// TIA Portal V15.1 export
// export: Created 2024-06-21T08:40:42.5093779Z, ExportSetting WithDefaults, DisplayName Totally Integrated Automation Portal, DisplayVersion V15.1 Update 5, DisplayName TIA Portal Openness, DisplayVersion V15.1 Update 5, DisplayName SINAMICS Startdrive Advanced, DisplayVersion V15.1, DisplayName G130, G150, S120, S150, SINAMICS MV, S210, DisplayVersion V15.1, DisplayName G110M, G120, G120C, G120D, G120P, DisplayVersion V15.1, DisplayName STEP 7 Professional, DisplayVersion V15.1 Update 5, DisplayName STEP 7 Safety, DisplayVersion V15.1, DisplayName WinCC Professional, DisplayVersion V15.1 Update 5, DisplayName SIMATIC Visualization Architect, DisplayVersion V15.1
DATA_BLOCK "_209000NCP01PNIODiag"   // DB270
{ S7_Optimized_Access := 'FALSE' }
AUTHOR : VCC
VERSION : 0.1
// stored: AutoNumber false, DBAccessibleFromOPCUA true, IsOnlyStoredInLoadMemory false, IsWriteProtectedInAS false
   VAR RETAIN
      "AD_209000AK01E1-BE30" { ExternalAccessible := 'False'; ExternalVisible := 'False'; ExternalWritable := 'False'} : Bool;   // Profinet device doesn't exist - PAC - Cabinet AK01 - node 30
      "AC_209000AE01-JC31" { ExternalAccessible := 'False'; ExternalVisible := 'False'; ExternalWritable := 'False'} : Bool;   // Profinet device doesn't exist - Gateway ETA Fuse - Cabinet AE01 - node 31
      "AC_209000AK02-JC32" { ExternalAccessible := 'False'; ExternalVisible := 'False'; ExternalWritable := 'False'} : Bool;   // Profinet device doesn't exist - Gateway ETA Fuse - Cabinet AK02 - node 32
      "AA_209000AK01-JW35" { ExternalAccessible := 'False'; ExternalVisible := 'False'; ExternalWritable := 'False'} : Bool;   // Profinet device doesn't exist - ET200sp I/O - Busnode AK01 - node 35
      "AA_209000AK03-JW36" { ExternalAccessible := 'False'; ExternalVisible := 'False'; ExternalWritable := 'False'} : Bool;   // Profinet device doesn't exist - ET200sp I/O - Busnode AK03 - node 36
      "AA_209000AK04-JW37" { ExternalAccessible := 'False'; ExternalVisible := 'False'; ExternalWritable := 'False'} : Bool;   // Profinet device doesn't exist - ET200sp I/O - Busnode AK04 - node 37
      "AA_209000AS01-JW38" { ExternalAccessible := 'False'; ExternalVisible := 'False'; ExternalWritable := 'False'} : Bool;   // Profinet device doesn't exist - ET200sp I/O - Busnode AS01 - node 38
      "AA_209000AS02-JW39" { ExternalAccessible := 'False'; ExternalVisible := 'False'; ExternalWritable := 'False'} : Bool;   // Profinet device doesn't exist - ET200sp I/O - Busnode AS02 - node 39
      "AA_209000AE02-JW208" { ExternalAccessible := 'False'; ExternalVisible := 'False'; ExternalWritable := 'False'} : Bool;   // Profinet device doesn't exist - PN/PN coupler - 209000 <-> 308210 AE02 - node 208
      "AA_209000AE02-JW210" { ExternalAccessible := 'False'; ExternalVisible := 'False'; ExternalWritable := 'False'} : Bool;   // Profinet device doesn't exist - Switch - Cabinet AE02 - node 210
      "AA_209000AE02-JW211" { ExternalAccessible := 'False'; ExternalVisible := 'False'; ExternalWritable := 'False'} : Bool;   // Profinet device doesn't exist - Switch - Cabinet AE02 - node 211
      "AA_211212AE1-JW200" { ExternalAccessible := 'False'; ExternalVisible := 'False'; ExternalWritable := 'False'} : Bool;   // Profinet device doesn't exist - ET200sp I/O - Busnode PLS211212AE1 - node 200
      "AC_209000AK01E1-BE30Fault" { ExternalAccessible := 'False'; ExternalVisible := 'False'; ExternalWritable := 'False'} : Bool;   // Faulty profinet device -> For more detail information look for N.A. alarms in the alarmlist - PAC - Cabinet AK01 - node 30
      "AC_209000AE01-JC31Fault" { ExternalAccessible := 'False'; ExternalVisible := 'False'; ExternalWritable := 'False'} : Bool;   // Faulty profinet device -> For more detail information look for N.A. alarms in the alarmlist - Gateway ETA Fuse - Cabinet AE01 - node 31
      "AC_209000AK02-JC32Fault" { ExternalAccessible := 'False'; ExternalVisible := 'False'; ExternalWritable := 'False'} : Bool;   // Faulty profinet device -> For more detail information look for N.A. alarms in the alarmlist - Gateway ETA Fuse - Cabinet AK02 - node 32
      "AC_209000AK01-JW35Fault" { ExternalAccessible := 'False'; ExternalVisible := 'False'; ExternalWritable := 'False'} : Bool;   // Faulty profinet device -> For more detail information look for N.A. alarms in the alarmlist - ET200sp I/O - Busnode AK01 - node 35
      "AC_209000AK03-JW36Fault" { ExternalAccessible := 'False'; ExternalVisible := 'False'; ExternalWritable := 'False'} : Bool;   // Faulty profinet device -> For more detail information look for N.A. alarms in the alarmlist - ET200sp I/O - Busnode AK03 - node 36
      "AC_209000AK04-JW37Fault" { ExternalAccessible := 'False'; ExternalVisible := 'False'; ExternalWritable := 'False'} : Bool;   // Faulty profinet device -> For more detail information look for N.A. alarms in the alarmlist - ET200sp I/O - Busnode AK04 - node 37
      "AC_209000AS01-JW38Fault" { ExternalAccessible := 'False'; ExternalVisible := 'False'; ExternalWritable := 'False'} : Bool;   // Faulty profinet device -> For more detail information look for N.A. alarms in the alarmlist - ET200sp I/O - Busnode AS01 - node 38
      "AC_209000AS02-JW39Fault" { ExternalAccessible := 'False'; ExternalVisible := 'False'; ExternalWritable := 'False'} : Bool;   // Faulty profinet device -> For more detail information look for N.A. alarms in the alarmlist - ET200sp I/O - Busnode AS02 - node 39
      "AC_209000AE02-JW208Fault" { ExternalAccessible := 'False'; ExternalVisible := 'False'; ExternalWritable := 'False'} : Bool;   // Faulty profinet device -> For more detail information look for N.A. alarms in the alarmlist - PN/PN coupler - 209000 <-> 308210 AE02 - node 208
      "AC_209000AE02-JW210Fault" { ExternalAccessible := 'False'; ExternalVisible := 'False'; ExternalWritable := 'False'} : Bool;   // Faulty profinet device -> For more detail information look for N.A. alarms in the alarmlist - Switch - Cabinet AE02 - node 210
      "AC_209000AE02-JW211Fault" { ExternalAccessible := 'False'; ExternalVisible := 'False'; ExternalWritable := 'False'} : Bool;   // Faulty profinet device -> For more detail information look for N.A. alarms in the alarmlist - Switch - Cabinet AE02 - node 211
      "AC_211212AE1-JW200Fault" { ExternalAccessible := 'False'; ExternalVisible := 'False'; ExternalWritable := 'False'} : Bool;   // Faulty profinet device -> For more detail information look for N.A. alarms in the alarmlist - ET200sp I/O - Busnode PLS211212AE1 - node 200
      AE_RefreshLists { ExternalAccessible := 'False'; ExternalVisible := 'False'; ExternalWritable := 'False'} : Bool;   // The information (Name - IP address - MAC address) from the profinet devices are not up-to-date / Info -> The information (Name - IP address - MAC address) from the profinet devices are not up-to-date
      "209000AK01-JW35AlarmABCondition" { ExternalAccessible := 'False'; ExternalVisible := 'False'; ExternalWritable := 'False'} : Bool;   // Alarm AB condition
      "209000AK03-JW36AlarmABCondition" { ExternalAccessible := 'False'; ExternalVisible := 'False'; ExternalWritable := 'False'} : Bool;   // Alarm AB condition
      "209000AK04-JW37AlarmABCondition" { ExternalAccessible := 'False'; ExternalVisible := 'False'; ExternalWritable := 'False'} : Bool;   // Alarm AB condition
      "209000AS01-JW38AlarmABCondition" { ExternalAccessible := 'False'; ExternalVisible := 'False'; ExternalWritable := 'False'} : Bool;   // Alarm AB condition
      "209000AS02-JW39AlarmABCondition" { ExternalAccessible := 'False'; ExternalVisible := 'False'; ExternalWritable := 'False'} : Bool;   // Alarm AB condition
      "209000AE02-JW208AlarmABCondition" { ExternalAccessible := 'False'; ExternalVisible := 'False'; ExternalWritable := 'False'} : Bool;   // Alarm AB condition
      "209000AE02-JW210AlarmABCondition" { ExternalAccessible := 'False'; ExternalVisible := 'False'; ExternalWritable := 'False'} : Bool;   // Alarm AB condition
      "209000AE02-JW211AlarmABCondition" { ExternalAccessible := 'False'; ExternalVisible := 'False'; ExternalWritable := 'False'} : Bool;   // Alarm AB condition
      "211212AE1-JW200AlarmABCondition" { ExternalAccessible := 'False'; ExternalVisible := 'False'; ExternalWritable := 'False'} : Bool;   // Alarm AB condition
      "H_209000AK01E1-BE30IAnim" : Word;   // HMI Animation of the icon
      "H_209000AE01-JC31IAnim" : Word;   // HMI Animation of the icon
      "H_209000AK02-JC32IAnim" : Word;   // HMI Animation of the icon
      "H_209000AK01-JW35IAnim" : Word;   // HMI Animation of the icon
      "H_209000AK03-JW36IAnim" : Word;   // HMI Animation of the icon
      "H_209000AK04-JW37IAnim" : Word;   // HMI Animation of the icon
      "H_209000AS01-JW38IAnim" : Word;   // HMI Animation of the icon
      "H_209000AS02-JW39IAnim" : Word;   // HMI Animation of the icon
      "H_209000AE02-JW208IAnim" : Word;   // HMI Animation of the icon
      "H_209000AE02-JW210IAnim" : Word;   // HMI Animation of the icon
      "H_209000AE02-JW211IAnim" : Word;   // HMI Animation of the icon
      "H_211212AE1-JW200IAnim" : Word;   // HMI Animation of the icon
      "H_209000AK01E1-BE30IAnim2" : Word;   // HMI Animation of the icon
      "H_209000AE01-JC31IAnim2" : Word;   // HMI Animation of the icon
      "H_209000AK02-JC32IAnim2" : Word;   // HMI Animation of the icon
      "H_209000AK01-JW35IAnim2" : Word;   // HMI Animation of the icon
      "H_209000AK03-JW36IAnim2" : Word;   // HMI Animation of the icon
      "H_209000AK04-JW37IAnim2" : Word;   // HMI Animation of the icon
      "H_209000AS01-JW38IAnim2" : Word;   // HMI Animation of the icon
      "H_209000AS02-JW39IAnim2" : Word;   // HMI Animation of the icon
      "H_209000AE02-JW208IAnim2" : Word;   // HMI Animation of the icon
      "H_209000AE02-JW210IAnim2" : Word;   // HMI Animation of the icon
      "H_209000AE02-JW211IAnim2" : Word;   // HMI Animation of the icon
      "H_211212AE1-JW200IAnim2" : Word;   // HMI Animation of the icon
      H_IAnim : Word;   // Icon Animation / Animation
      H_Anim : Word;   // Animation
      H_DBnr : Int;   // DB number
      H_HMICmd : Word;   // HMI Command
      HMICmdResetPNStatus { ExternalAccessible := 'False'; ExternalVisible := 'False'; ExternalWritable := 'False'} : Bool;   // HMI Command - Reset Profinet Status
      HMICmdRefreshPNInfo { ExternalAccessible := 'False'; ExternalVisible := 'False'; ExternalWritable := 'False'} : Bool;   // HMI Command - Refresh Profinet Information (Name - IP address - MAC address)
      AlarmA { ExternalAccessible := 'False'; ExternalVisible := 'False'; ExternalWritable := 'False'} : Bool;   // Alarm A
      AlarmB { ExternalAccessible := 'False'; ExternalVisible := 'False'; ExternalWritable := 'False'} : Bool;   // Alarm B
      AlarmC { ExternalAccessible := 'False'; ExternalVisible := 'False'; ExternalWritable := 'False'} : Bool;   // Alarm C
      AlarmD { ExternalAccessible := 'False'; ExternalVisible := 'False'; ExternalWritable := 'False'} : Bool;   // Alarm D
      AlarmABCondition { ExternalAccessible := 'False'; ExternalVisible := 'False'; ExternalWritable := 'False'} : Bool;   // Alarm AB conditon
   END_VAR
BEGIN
END_DATA_BLOCK
